
// ===== library: MasterCopy "Copy of Program blocks in MTConnect" =====
// protected blocks, not shown: "MTCONNECT", "TimeStamp"

// folder: MTConnect

DATA_BLOCK "MTCData"   // DB4
{ S7_Optimized_Access := 'TRUE' }
VERSION : 0.1
   VAR
      "Bool" : Array[0..1] of "DataItemBool";
      Numeric : Array[0..1] of "DataItemNumeric";
      "String" : Array[0..1] of "DataItemString";
   END_VAR
BEGIN
   "Bool"[0]."name" := 'estop';
   "Bool"[0].category := 1;   // 1) EVENT 2) SAMPLE 3)CONDITION
   "Bool"[1]."name" := 'btag1';
   "Bool"[0].value := FALSE;
   "Bool"[0].prevValue := FALSE;
   "Bool"[0].send := FALSE;
   "Bool"[1].category := 0;
   "Bool"[1].value := FALSE;
   "Bool"[1].prevValue := FALSE;
   "Bool"[1].send := FALSE;
   Numeric[0]."name" := 'cycles';
   Numeric[0].category := 0;
   Numeric[0].value := 0.0;
   Numeric[0].prevvalue := 0.0;
   Numeric[0].send := FALSE;
   Numeric[1]."name" := 'ftag1';
   Numeric[1].category := 0;
   Numeric[1].value := 0.0;
   Numeric[1].prevvalue := 0.0;
   Numeric[1].send := FALSE;
END_DATA_BLOCK

FUNCTION "SizeOf" : Int   // FC4, SCL
{ S7_Optimized_Access := 'TRUE' }
VERSION : 0.1
   VAR_INPUT
      Arrayin : Variant;
   END_VAR
   VAR_TEMP
      erro : Int;
   END_VAR
BEGIN
   #SizeOf := CountOfElements(#Arrayin);
END_FUNCTION